// SIMATIC S7-200 project (STEP 7-Micro/WIN), CPU 222 REL 01.22

SYMBOL_TABLE USUARIO1
FR1              I0.0     // RELE TERMICO
S1               I0.1     // PULSDOR PARO
S2               I0.2     // PULSADOR MARCHA DERECHA
S3               I0.3     // `PULSADOR MARCHA IZQUIERDAA
KM1              Q0.0     // CONTACTOR MARCHA DERECHA
H1               Q0.1     // SEÑALIZACION MARCHA DERECHA
KM2              Q0.2     // CONTACTOR MARCHA IZQUIERDA
H2               Q0.3     // SEÑALIZACION MARCHA IZQUIERDA
H3               Q0.4     // SEÑALIZACION AVERIA
H4               Q0.5     // SEÑALIZACION PARADA
END_SYMBOL_TABLE

ORGANIZATION_BLOCK PRINCIPAL:OB1
TITLE=COMENTARIOS DEL PROGRAMA
BEGIN
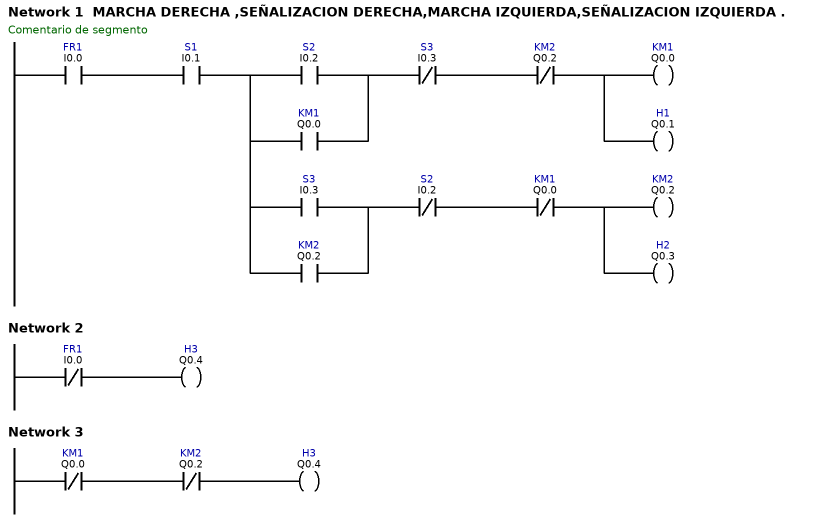
Network 1 // MARCHA DERECHA ,SEÑALIZACION DERECHA,MARCHA IZQUIERDA,SEÑALIZACION IZQUIERDA
.
// Comentario de segmento
LD     FR1:I0.0
A      S1:I0.1
LPS
LD     S2:I0.2
O      KM1:Q0.0
AN     S3:I0.3
AN     KM2:Q0.2
ALD
=      KM1:Q0.0
=      H1:Q0.1
LPP
LD     S3:I0.3
O      KM2:Q0.2
AN     S2:I0.2
AN     KM1:Q0.0
ALD
=      KM2:Q0.2
=      H2:Q0.3
Network 2
LDN    FR1:I0.0
=      H3:Q0.4
Network 3
LDN    KM1:Q0.0
AN     KM2:Q0.2
=      H3:Q0.4
END_ORGANIZATION_BLOCK
